{attribute 'qualified_only'}
//joints parameters of slave arms
VAR_GLOBAL 	
	// absolute encoder value at minimal joint positon
	g_minLinkEncoder :ARRAY[1..g_sArmNum, 1..g_sJntNum] OF DINT;
		 
	// absolute encoder value at maximum joint positon
	g_maxLinkEncoder :ARRAY[1..g_sArmNum, 1..g_sJntNum] OF DINT;
	
	// absolute encoder value at calibrated positon
	g_caliLinkEncoder :ARRAY[1..g_sArmNum, 1..g_sJntNum] OF DINT;
	
	 // if absolute encoder value cross zeros within joint motion range
	 // NOTICE: joint 7 is always 0.
	g_linkEncZeroCross :ARRAY[1..g_sArmNum, 1..g_sJntNum] OF INT;
		 
	 // joint SDO address
	//g_slaveArmNetID: ARRAY[1..4] OF T_AmsNetId:=['169.254.223.120.10.1','192.168.2.91.4.1','192.168.2.91.6.1','192.168.2.91.5.1'];
	//g_slaveJointNetPort:ARRAY[1..g_sArmNum,1..g_sJntNum] OF UINT :=[
	//	1005,	1006,	1007,	2(1008),	3(1009),
	//	1005,	1006,	1007,	2(1008),	3(1009),
	//	1005,	1006,	1007,	2(1008),	3(1009),
	//	1005,	1006,	1007,	2(1008),	3(1009)];
	//g_slaveLEDNetPort:ARRAY[1..g_sArmNum] OF UINT :=[4(1003)];
		
//################ DO NOT modify parameters below ###########################
	// abolute encoder expanded limit buffer in case there is calibrtion error at limit position
	g_linkEncLimitBuffer :ARRAY [1..g_sJntNum] OF DINT := [2(1000),6(1000)];
	
	// absolute encoder direction
	g_asbEncoderDir :ARRAY[1..g_sJntNum] OF INT :=[-1, 1, 1, -1, -1, -1, -1, -1];
	
	// flag if joint can rotate multiple cycles
	g_multipleCyclesJoint :ARRAY[1..g_sArmNum, 1..g_sJntNum] OF INT :=
		[0, 0, 0, 1, 1, 1, 1, 1,
		 0, 0, 0, 1, 1, 1, 1, 1,
		 0, 0, 0, 1, 1, 1, 1, 1,
		 0, 0, 0, 1, 1, 1, 1, 1];
		 
	// joint position at link encoder calibrated point
	g_linkEncCaliJntPos :ARRAY[1..g_sJntNum] OF LREAL :=
		[0.0,-pi/2, 0.54608, 5(-pi/2)];
	g_linkJntPosOffset:ARRAY[1..g_sArmNum, 1..g_sJntNum] OF LREAL :=
	[0, 0, 0, 0, 0, 0, 0, 0,
	 0, 0, 0, 0, 0, 0, 0, 0,
	 0, 0, 0, 0, 0, 0, 0, 0,
	 0, 0, 0, 0, 0, 0, 0, 0];
	
END_VAR

(* stored: Version 1.1.0.1, ProductVersion 3.1.4024.11
   GVL GVL_SlaveJointEncoderCaliData: Id {7eae507e-05dd-426e-b2d5-321e9d64d4f5} *)
